(* CODESYS project I2C_UBrain1.library
   Description: Library containing device support for BRian1 under Raspberry Pi
   Author: OOO ASU L
   Version: 1.1.0.0
   Company: OOO ASU
   Title: Raspberry I2C Brian1
   DefaultNamespace: BRAIN1
   Placeholder: PlaceholderTemplate

Project tree, tasks and I/O mapping:
  libraries: Standard, * (System); IoStandard, * (System); Raspberry Pi Peripherals, * (3S - Smart Software Solutions GmbH)
  function block UBrainDIO [ST]: AfterReadInputs, BeforeWriteOutputs
  00000000-0000-0000-0000-000000000000|D:\CoDeSys\LibrariesV3\trunk\Intern\CAA\CAA Template\3.4.0.0 draft\Placeholder.xml
  00000000-0000-0000-0000-000000000000|D:\CoDeSys\LibrariesV3\trunk\Intern\CAA\CAA Template\3.2.0.3 draft\Prefix.pdf
  00000000-0000-0000-0000-000000000000|D:\CoDeSys\LibrariesV3\trunk\Intern\CAA\CAA Template\3.5.2.0 draft\Placeholder.xml
*)

// UBrainDIO
FUNCTION_BLOCK UBrainDIO EXTENDS i2c
VAR_INPUT
	bDOut1 : BYTE := 0;
	bColorButton : ARRAY [0..8] OF BYTE ;
END_VAR
VAR_OUTPUT
	bDin1 : BYTE := 0;
	bButtons : BYTE := 0;
	xValidRead : BOOL := FALSE;
	xValidWrite : BOOL := FALSE;
END_VAR
VAR
	timerR: TON := (IN:=TRUE);
	timerW: TON := (IN:=TRUE);
	
END_VAR
VAR CONSTANT
		
	// Направление: true - передача, false- приём
	directTX: BOOL := true;
END_VAR

//xNewMeasurement := FALSE;

SUPER^();

CASE _iState OF
0:
	IF usiAddress = 0 THEN
		usiAddress := 16#72;
	END_IF
	IF SUPER^.init() THEN
		_iState := 5;
	END_IF	

5:	
	TimerR.pt := T#50MS;
	TimerW.pt := T#50MS;
	_iState := 10;	
	xValidRead := FALSE;
	xValidWrite := FALSE;
END_CASE

METHOD AfterReadInputs : INT
VAR
	Buffer : ARRAY[0..2] OF BYTE;
	len: dINT;
END_VAR
SUPER^.AfterReadInputs();

IF _iState = 10 THEN
	timerR(IN:=TRUE);
	IF timerR.Q THEN
		Buffer[0] := 16#0F;//BOOL_TO_BYTE(NOT directTX);	
		len := Write(ADR(Buffer), 1);
		IF len = 1 THEN
			len := Read(ADR(Buffer), 2);
			IF len = 2 THEN
				bDin1 := Buffer[0];
				bButtons := Buffer[1];
	//			xNewMeasurement := TRUE;
				xValidRead := TRUE;
			ELSE
				xValidRead := FALSE;
			END_IF
		ELSE
			xValidRead := FALSE;	
		END_IF
			
			
//		Write8(0, 16#51);	//new measurement
		timerR(IN:=FALSE);
	END_IF		
END_IF
END_METHOD

METHOD BeforeWriteOutputs : INT
VAR
	Buffer2 : ARRAY[0..8] OF BYTE;
	len: dINT;
END_VAR
SUPER^.BeforeWriteOutputs();

IF _iState = 10 THEN
	timerW(IN:=TRUE);
	IF timerW.Q THEN	
//		Buffer[0] := bDOut1;
//		Buffer[1] := bColorButton1;
//		Buffer[2] := bColorButton2;
//		Buffer[3] := bColorButton3;
//		Buffer[4] := bColorButton4;
//		Buffer[5] := bColorButton5;
//		Buffer[6] := bColorButton6;
//		Buffer[7] := bColorButton7;
//		Buffer[8] := bColorButton8;
		
		
		Buffer2[0] := 16#F0; //BOOL_TO_BYTE(directTX);	
		len := Write(ADR(Buffer2), 1);
		IF len = 1  THEN
			Buffer2[0] := bColorButton[0];
			Buffer2[1] := bColorButton[1];
			Buffer2[2] := bColorButton[2];
			Buffer2[3] := bColorButton[3];
			Buffer2[4] := bColorButton[4];
			Buffer2[5] := bColorButton[5];
			Buffer2[6] := bColorButton[6];
			Buffer2[7] := bColorButton[7];
			Buffer2[8] := bDOut1;
			len := Write(ADR(Buffer2), 9);
			IF len = 9 THEN
				xValidWrite := TRUE;
			ELSE
				xValidWrite := FALSE;
			END_IF
		ELSE
			xValidWrite := FALSE;
		END_IF
			
		timerW(IN:=FALSE);
	END_IF		
END_IF
END_METHOD

END_FUNCTION_BLOCK
